INTERFACE I_DriveAxisCmds EXTENDS I_OUTPUTS

PROPERTY CommandHalt : BOOL
SET
END_SET
END_PROPERTY

PROPERTY CommandMoveAbsolute : BOOL
SET
END_SET
END_PROPERTY

PROPERTY CommandMoveHome : BOOL
SET
END_SET
END_PROPERTY

METHOD ErrorHandling
VAR_INPUT
END_VAR
END_METHOD

(*
    Check all post condition before updating bCommandedMoveAbsolute
    The implmentatation will depend on the axis type
    DS402 NC/Direct axis : Implementation need to check that the drive is in the correct mode before initaiting the move then set bCommandedMoveAbsolute
    MP NC axis : will immediately write to bCommandedMoveAbsolute
*)
METHOD StartMove : BOOL
VAR_INPUT
	MoveMode	: E_EpicsMotorCmd;
	CmdExecute	: BOOL;
END_VAR
END_METHOD

END_INTERFACE

(* stored: Version 1.1.0.1
   Itf I_DriveAxisCmds: Id {6c0355c5-d46f-449f-8c34-fd9a1ef64ba8}
   Property CommandHalt: Id {28caa621-b1b5-45c3-948b-355529ae63c2}
   Set Set: Id {afbd26a2-5d4f-4673-a5ff-92792f920642}
   Property CommandMoveAbsolute: Id {be1022ab-c175-45cf-b747-4904f7dbb61a}
   Set Set: Id {148eb03e-69c6-4884-b363-b91c6e29515e}
   Property CommandMoveHome: Id {c447ca24-e237-4885-a9a3-281864c8338b}
   Set Set: Id {fd07a648-391b-4835-a127-b5f46d9080b8}
   Method ErrorHandling: Id {8c3f2673-8367-4245-8039-269c7637bb4c}
   Method StartMove: Id {2d898c45-221d-4ab1-9add-83136ca35be3} *)
